// Copyright (c) 2024 Loupe (https://loupe.team), provided under the MIT License.
{attribute 'qualified_only'}
{attribute 'strict'}
TYPE ABBLINKIN_COMMAND_TYPE :
(
	GET_IO,
	GET_CTRL_STATE,
	GET_OP_MODE,
	GET_RAPID_STATE,
	GET_SYMBOL,
	POWER_OFF,
	POWER_ON,
	RAPID_RESET,
	RAPID_START,
	RAPID_STOP,
	SET_IO,
	SET_SYMBOL
);
END_TYPE

(* stored: Version 1.1.0.1, ProductVersion 3.1.4024.12
   DUT ABBLINKIN_COMMAND_TYPE: Id {d7d89884-2a0b-4df0-8653-de60d8f0522a} *)
